(*
SPDX-FileCopyrightText: © 2026 Oleksandr Tiutyk <trofimich@gmail.com>
SPDX-License-Identifier: MIT
License: https://opensource.org/license/mit
*)

INTERFACE IReadOnlyTrafficLight EXTENDS TOF_Automation.ICompositeAutomationComponent, TOF_Core.IIOBindable

{attribute 'monitoring' := 'call'}
PROPERTY FINAL ActiveLight : TRAFFIC_LIGHT_COLOR
GET
END_GET
END_PROPERTY

{attribute 'monitoring' := 'call'}
PROPERTY FINAL GreenLight : TOF_Devices_IO.IReadOnlyDigitalOutput
GET
END_GET
END_PROPERTY

{attribute 'monitoring' := 'call'}
PROPERTY FINAL RedLight : TOF_Devices_IO.IReadOnlyDigitalOutput
GET
END_GET
END_PROPERTY

{attribute 'monitoring' := 'call'}
PROPERTY FINAL YellowLight : TOF_Devices_IO.IReadOnlyDigitalOutput
GET
END_GET
END_PROPERTY

END_INTERFACE

(* stored: Version 1.1.0.1
   Itf IReadOnlyTrafficLight: Id {a8df015d-8922-495a-ad01-cfd3bf7b73ee}
   Folder Statuses: Id {60b1587b-885f-462b-9258-c0032b67e1b8}
   Folder SubDevices: Id {03444497-d774-43df-a0a2-1c95d95ddae7}
   Property ActiveLight: Id {22a271f2-6628-443b-bcc3-2a9d13167870}
   Get Get: Id {49a6a85e-cb13-4078-962d-97d6fd689dea}
   Property GreenLight: Id {19fb6575-5b8b-4060-a1a1-95f5e6566b6d}
   Get Get: Id {deae0774-8088-42bc-8629-a02b0a46cb68}
   Property RedLight: Id {679ee5d4-5cb8-4c95-b31e-a55fc8919ccc}
   Get Get: Id {223e3e3f-34d8-4436-8942-de97addbd869}
   Property YellowLight: Id {04ddbedb-0c4e-4afd-b5c7-ca4a99aaa07f}
   Get Get: Id {85d1400d-f74b-4ccc-98b7-d62daa9bfc5c} *)
